# EPICS autosave request: LabJackApp/Db/LabJack_T7_settings.req
# Digital Inputs
$(P)LJT7:$(N):DI0.DESC
$(P)LJT7:$(N):DI1.DESC
$(P)LJT7:$(N):DI2.DESC
$(P)LJT7:$(N):DI3.DESC
$(P)LJT7:$(N):DI4.DESC
$(P)LJT7:$(N):DI5.DESC
$(P)LJT7:$(N):DI6.DESC
$(P)LJT7:$(N):DI7.DESC
$(P)LJT7:$(N):DI8.DESC
$(P)LJT7:$(N):DI9.DESC
$(P)LJT7:$(N):DI10.DESC
$(P)LJT7:$(N):DI11.DESC

# Digital Outputs
$(P)LJT7:$(N):DO0.DESC
$(P)LJT7:$(N):DO0
$(P)LJT7:$(N):DO1.DESC
$(P)LJT7:$(N):DO1
$(P)LJT7:$(N):DO2.DESC
$(P)LJT7:$(N):DO2
$(P)LJT7:$(N):DO3.DESC
$(P)LJT7:$(N):DO3
$(P)LJT7:$(N):DO4.DESC
$(P)LJT7:$(N):DO4
$(P)LJT7:$(N):DO5.DESC
$(P)LJT7:$(N):DO5
$(P)LJT7:$(N):DO6.DESC
$(P)LJT7:$(N):DO6
$(P)LJT7:$(N):DO7.DESC
$(P)LJT7:$(N):DO7
$(P)LJT7:$(N):DO8.DESC
$(P)LJT7:$(N):DO8
$(P)LJT7:$(N):DO9.DESC
$(P)LJT7:$(N):DO9
$(P)LJT7:$(N):DO10.DESC
$(P)LJT7:$(N):DO10

# Analog Inputs
$(P)LJT7:$(N):AI0.DESC
$(P)LJT7:$(N):AI0.SCAN
$(P)LJT7:$(N):AI1.DESC
$(P)LJT7:$(N):AI1.SCAN
$(P)LJT7:$(N):AI2.DESC
$(P)LJT7:$(N):AI2.SCAN
$(P)LJT7:$(N):AI3.DESC
$(P)LJT7:$(N):AI3.SCAN
$(P)LJT7:$(N):AI4.DESC
$(P)LJT7:$(N):AI4.SCAN
$(P)LJT7:$(N):AI5.DESC
$(P)LJT7:$(N):AI5.SCAN
$(P)LJT7:$(N):AI6.DESC
$(P)LJT7:$(N):AI6.SCAN
$(P)LJT7:$(N):AI7.DESC
$(P)LJT7:$(N):AI7.SCAN
$(P)LJT7:$(N):AI8.DESC
$(P)LJT7:$(N):AI8.SCAN
$(P)LJT7:$(N):AI9.DESC
$(P)LJT7:$(N):AI9.SCAN
$(P)LJT7:$(N):AI10.DESC
$(P)LJT7:$(N):AI10.SCAN
$(P)LJT7:$(N):AI11.DESC
$(P)LJT7:$(N):AI11.SCAN
$(P)LJT7:$(N):AI12.DESC
$(P)LJT7:$(N):AI12.SCAN
$(P)LJT7:$(N):AI13.DESC
$(P)LJT7:$(N):AI13.SCAN

# AI Configuration
$(P)LJT7:$(N):seDiff_Ch0
$(P)LJT7:$(N):seDiff_Ch2
$(P)LJT7:$(N):seDiff_Ch4
$(P)LJT7:$(N):seDiff_Ch6
$(P)LJT7:$(N):seDiff_Ch8
$(P)LJT7:$(N):seDiff_Ch10
$(P)LJT7:$(N):seDiff_Ch12
$(P)LJT7:$(N):AIRange0
$(P)LJT7:$(N):AIRange1
$(P)LJT7:$(N):AIRange2
$(P)LJT7:$(N):AIRange3
$(P)LJT7:$(N):AIRange4
$(P)LJT7:$(N):AIRange5
$(P)LJT7:$(N):AIRange6
$(P)LJT7:$(N):AIRange7
$(P)LJT7:$(N):AIRange8
$(P)LJT7:$(N):AIRange9
$(P)LJT7:$(N):AIRange10
$(P)LJT7:$(N):AIRange11
$(P)LJT7:$(N):AIRange12
$(P)LJT7:$(N):AIRange13
$(P)LJT7:$(N):AIResolution0
$(P)LJT7:$(N):AIResolution1
$(P)LJT7:$(N):AIResolution2
$(P)LJT7:$(N):AIResolution3
$(P)LJT7:$(N):AIResolution4
$(P)LJT7:$(N):AIResolution5
$(P)LJT7:$(N):AIResolution6
$(P)LJT7:$(N):AIResolution7
$(P)LJT7:$(N):AIResolution8
$(P)LJT7:$(N):AIResolution9
$(P)LJT7:$(N):AIResolution10
$(P)LJT7:$(N):AIResolution11
$(P)LJT7:$(N):AIResolution12
$(P)LJT7:$(N):AIResolution13

# Analog Outputs
$(P)LJT7:$(N):AO0.DESC
$(P)LJT7:$(N):AO0
$(P)LJT7:$(N):AO0TweakVal
$(P)LJT7:$(N):AO1.DESC
$(P)LJT7:$(N):AO1
$(P)LJT7:$(N):AO1TweakVal
